// TIA Portal V18 export
DATA_BLOCK "Metering control"   // DB116
{ S7_Optimized_Access := 'TRUE' }
VERSION : 0.1
// stored: AutoNumber true, DBAccessibleFromOPCUA true, IsOnlyStoredInLoadMemory false, IsRetainMemResEnabled false, IsWriteProtectedInAS false, MemoryReserve 100
   VAR RETAIN
      "outlet valve" : Struct
         selection : Int;
         "common selected" : Bool;
         individual : Bool;
      END_STRUCT;
      Reneration : Struct
         selection : Int := 1;
         selected : Bool;
      END_STRUCT;
      Flush : Struct
         selection : Int;
         selected : Bool;
      END_STRUCT;
      compression : Struct
         selection : Int;
         selected : Bool;
      END_STRUCT;
      Refilling : Struct
         "selection A" : Int;
         "selection B" : Int;
      END_STRUCT;
      "system Preparation" : Struct
         "A selection" : Int := 1;
         "B selection" : Int := 1;
      END_STRUCT;
      "Ready to meter" : Struct
         "pressure less selection A" : Int := 1;
         "Pressure less selection  B" : Int := 1;
         "Heater interlock" : Bool;
      END_STRUCT;
   END_VAR
BEGIN
END_DATA_BLOCK
